FUNCTION_BLOCK FB_WriteAmsValue
VAR_INPUT
	tUpdate					:	TIME 				:=T#900MS;
	
	sNetId					:	T_AmsNetId			:='';
	nPort					:	T_AmsPort			:=851;
	sVarName				:	STRING(255)			:='';
	nSrcAddr				:	PVOID;
	nSrcLen					:	UDINT;
	tWriteTimeout			:	TIME				:=T#2000MS;
	
END_VAR

VAR_OUTPUT
END_VAR

VAR
	
	bWriteError			: BOOL := FALSE;
	nWriteErrorId		: UDINT;
	PT_Write			: TIME := T#5S;
	
	ET_Write			: TIME := T#0MS;
	bReadEnable			: BOOL := FALSE;
	bWriteBusy			: BOOL := FALSE;
	
	TON_Write		: TON;
	FB_writer		: FB_WriteAdsSymByName;
END_VAR

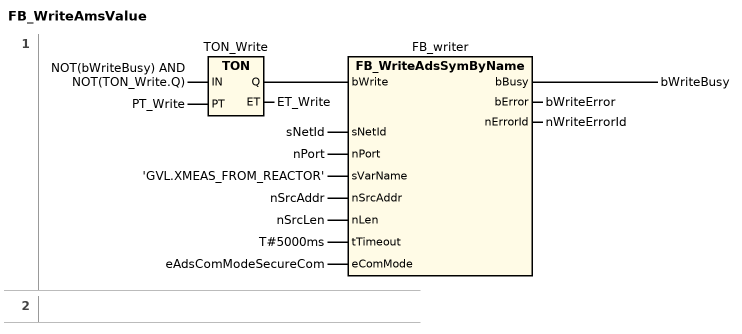
// NETWORK 1
TON_Write(IN := NOT(bWriteBusy) AND NOT(TON_Write.Q), PT := PT_Write, ET => ET_Write); // TON
FB_writer(
    bWrite := TON_Write.Q,
    sNetId := sNetId,
    nPort := nPort,
    sVarName := 'GVL.XMEAS_FROM_REACTOR',
    nSrcAddr := nSrcAddr,
    nLen := nSrcLen,
    tTimeout := T#5000ms,
    eComMode := eAdsComModeSecureCom,
    bError => bWriteError,
    nErrorId => nWriteErrorId); // FB_WriteAdsSymByName
bWriteBusy := FB_writer.bBusy;

// NETWORK 2

END_FUNCTION_BLOCK

(* stored: Version 1.1.0.1, ProductVersion 3.1.4024.11
   POU FB_WriteAmsValue: Id {f1b6e663-da5e-4f67-95a9-68e2c44d06ae}, SpecialFunc None *)
